FUNCTION_BLOCK ONE_CLASS_SVM
  {SET_ATTRIBUTE(OpcUa, SERVICE)}
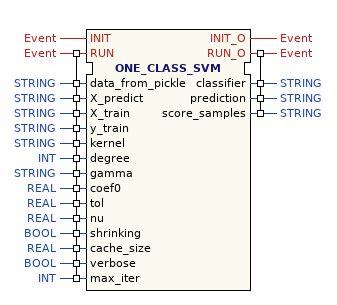
  EVENT_INPUT
    INIT;
    RUN WITH data_from_pickle, X_predict, X_train, y_train, kernel, degree, gamma, coef0, tol, nu, shrinking, cache_size, verbose, max_iter; {SET_ATTRIBUTE(OpcUa, Method)}
  END_EVENT
  EVENT_OUTPUT
    INIT_O;
    RUN_O WITH classifier, prediction, score_samples;
  END_EVENT
  VAR_INPUT
    data_from_pickle : STRING; {SET_ATTRIBUTE(OpcUa, Variable.RUN)}
    X_predict : STRING; {SET_ATTRIBUTE(OpcUa, Variable.RUN)}
    X_train : STRING; {SET_ATTRIBUTE(OpcUa, Variable.RUN)}
    y_train : STRING; {SET_ATTRIBUTE(OpcUa, Variable.RUN)}
    kernel : STRING; {SET_ATTRIBUTE(OpcUa, Variable.RUN)}
    degree : INT; {SET_ATTRIBUTE(OpcUa, Variable.RUN)}
    gamma : STRING; {SET_ATTRIBUTE(OpcUa, Variable.RUN)}
    coef0 : REAL; {SET_ATTRIBUTE(OpcUa, Variable.RUN)}
    tol : REAL; {SET_ATTRIBUTE(OpcUa, Variable.RUN)}
    nu : REAL; {SET_ATTRIBUTE(OpcUa, Variable.RUN)}
    shrinking : BOOL; {SET_ATTRIBUTE(OpcUa, Variable.RUN)}
    cache_size : REAL; {SET_ATTRIBUTE(OpcUa, Variable.RUN)}
    verbose : BOOL; {SET_ATTRIBUTE(OpcUa, Variable.RUN)}
    max_iter : INT; {SET_ATTRIBUTE(OpcUa, Variable.RUN)}
  END_VAR
  VAR_OUTPUT
    classifier : STRING; {SET_ATTRIBUTE(OpcUa, Variable.RUN)}
    prediction : STRING; {SET_ATTRIBUTE(OpcUa, Variable.RUN)}
    score_samples : STRING; {SET_ATTRIBUTE(OpcUa, Variable.RUN)}
  END_VAR
END_FUNCTION_BLOCK
